(* IEC 61131-3 sources: ATCMcontrol_Engineering/src/COM/softing/fc/AddOns/Softing/4CPCTarget/Libs/ATCM_IEC1131_3/table_36, 9 files *)

(* ---- ctd.st ---- *)
(*[[
    UserURL= "ATCM:CTD_DINT.htm"
]]*)
(*
 *  IEC-1131-3 Standard Functionblock CTD for data type INT
 *  Purpose: Down Counter
 *)
FUNCTION_BLOCK CTD
VAR_INPUT  (* Inputs *)
    CD         : BOOL R_EDGE; (* count down if rising edge     *)
    LD         : BOOL;        (* if true, copy PV to CV        *)
    PV         : INT;         (* start value                   *)
END_VAR
VAR_OUTPUT (* Outputs *)
    Q          : BOOL;        (* TRUE if CV <= 0               *)
    CV         : INT;         (* counter output                *)
END_VAR

;(* add target specific implementation here *)

END_FUNCTION_BLOCK

(* ---- ctd_dint.st ---- *)
(*[[
    UserURL= "ATCM:CTD_DINT.htm"
]]*)
(*
 *  IEC-1131-3 Standard Functionblock CTD for data type DINT
 *  Purpose: Down Counter
 *)
FUNCTION_BLOCK CTD_DINT
VAR_INPUT  (* Inputs *)
    CD         : BOOL R_EDGE; (* count down if rising edge     *)
    LD         : BOOL;        (* if true, copy PV to CV        *)
    PV         : DINT;        (* start value                   *)
END_VAR
VAR_OUTPUT (* Outputs *)
    Q          : BOOL;        (* TRUE if CV <= 0               *)
    CV         : DINT;        (* counter output                *)
END_VAR

  IF LD THEN
	CV := PV;
  ELSIF CD AND (CV > FC_MIN_DINT) THEN
	CV:=CV-1;
  END_IF;

  Q := (CV <= 0);

END_FUNCTION_BLOCK

(* ---- ctd_dint_ex.st ---- *)
(*[[
    UserURL= "ATCM:CTD_DINT_EX.htm"
]]*)
(*
 *  IEC-1131-3 Standard Functionblock CTD for data type DINT
 *  Purpose: Down Counter with visualisation scaling parameters
 *)
FUNCTION_BLOCK CTD_DINT_EX
VAR_INPUT  (* Inputs *)
    CD         : BOOL R_EDGE; (* count down if rising edge     *)
    LD         : BOOL;        (* if true, copy PV to CV        *)
    PV         : DINT;        (* start value                   *)
END_VAR
VAR_INPUT  (* Parameters *)
    SCALEMIN   : DINT:=0;     (* minimum of scaling            *)
    SCALEMAX   : DINT:=100;   (* maximum of scaling            *)
END_VAR
VAR_OUTPUT (* Outputs *)
    Q          : BOOL;        (* TRUE if CV <= 0               *)
    CV         : DINT;        (* counter output                *)
    ERROR      : DINT;        (* error                         *)
END_VAR

ERROR := 0;
IF (SCALEMIN >= SCALEMAX) THEN
   ERROR:=-1;
END_IF;

IF LD THEN
   CV := PV;
ELSIF CD AND (CV > FC_MIN_DINT) THEN
   CV:=CV-1;
END_IF;

Q := (CV <= 0);

END_FUNCTION_BLOCK

(* ---- ctu.st ---- *)
(*[[
    UserURL= "ATCM:CTU_DINT.htm"
]]*)
(*
 *  IEC-1131-3 Standard Functionblock CTU for data type INT
 *  Purpose: Up Counter
 *)
FUNCTION_BLOCK CTU
VAR_INPUT (* Inputs *)
    CU         : BOOL R_EDGE; (* count up if rising edge *)
    R          : BOOL;        (* if true,  CV to zero    *)
    PV         : INT;         (* end value               *)
END_VAR
VAR_OUTPUT (* Outputs *)
    Q          : BOOL;        (* TRUE if CV >= PV        *)
    CV         : INT;         (* counter output          *)
END_VAR

;(* add target specific implementation here *)

END_FUNCTION_BLOCK

(* ---- ctu_dint.st ---- *)
(*[[
    UserURL= "ATCM:CTU_DINT.htm"
]]*)
(*
 *  IEC-1131-3 Standard Functionblock CTU for data type DINT
 *  Purpose: Up Counter
 *)
FUNCTION_BLOCK CTU_DINT
VAR_INPUT (* Inputs *)
    CU         : BOOL R_EDGE; (* count up if rising edge *)
    R          : BOOL;        (* if true,  CV to zero    *)
    PV         : DINT;        (* end value               *)
END_VAR
VAR_OUTPUT (* Outputs *)
    Q          : BOOL;        (* TRUE if CV >= PV        *)
    CV         : DINT;        (* counter output          *)
END_VAR

  IF R THEN
	CV := 0;
  ELSIF CU AND (CV < FC_MAX_DINT) THEN
	CV:=CV+1;
  END_IF;

  Q := (CV >= PV);

END_FUNCTION_BLOCK

(* ---- ctu_dint_ex.st ---- *)
(*[[
    UserURL= "ATCM:CTU_DINT_EX.htm"
]]*)
(*
 *  IEC-1131-3 Standard Functionblock CTU for data type DINT
 *  Purpose: Up Counter with visualisation scaling parameters
 *)
FUNCTION_BLOCK CTU_DINT_EX
VAR_INPUT  (* Inputs *)
    CU         : BOOL R_EDGE; (* count up if rising edge *)
    R          : BOOL;        (* if true,  CV to zero    *)
    PV         : DINT;        (* end value               *)
END_VAR
VAR_INPUT  (* Parameters *)
    SCALEMIN   : DINT:=0;     (* minimum of scaling      *)
    SCALEMAX   : DINT:=100;   (* maximum of scaling      *)
END_VAR
VAR_OUTPUT (* Outputs *)
    Q          : BOOL;        (* TRUE if CV >= PV        *)
    CV         : DINT;        (* counter output          *)
    ERROR      : DINT;        (* error                   *)
END_VAR

ERROR := 0;
IF (SCALEMIN >= SCALEMAX) THEN
    ERROR:=-1;
END_IF;

IF R THEN
    CV := 0;
ELSIF CU AND (CV < FC_MAX_DINT) THEN
    CV:=CV+1;
END_IF;

Q := (CV >= PV);

END_FUNCTION_BLOCK

(* ---- ctud.st ---- *)
(*[[
    UserURL= "ATCM:ctud_dint.htm"
]]*)
(*
 *  IEC-1131-3 Standard Functionblock CTUD for data type INT
 *  Purpose: Up/Down Counter
 *)
FUNCTION_BLOCK CTUD
VAR_INPUT (* Inputs *)
    CU         : BOOL R_EDGE; (* count up if rising edge   *)
    CD         : BOOL R_EDGE; (* count down if rising edge *)
    R          : BOOL;        (* Reset, set CV to 0        *)
    LD         : BOOL;        (* if true, copy PV to CV    *)
    PV         : INT;         (* start value               *)
END_VAR
VAR_OUTPUT (* Outputs *)
    QU         : BOOL;        (* TRUE if CV >= PV          *)
    QD         : BOOL;        (* TRUE if CV <= 0           *)
    CV         : INT;         (* counter output            *)
END_VAR

;(* add target specific implementation here *)

END_FUNCTION_BLOCK

(* ---- ctud_dint.st ---- *)
(*[[
    UserURL= "ATCM:CTUD_DINT.htm"
]]*)
(*
 *  IEC-1131-3 Standard Functionblock CTUD for data type DINT
 *  Purpose: Up/Down Counter
 *)
FUNCTION_BLOCK CTUD_DINT
VAR_INPUT (* Inputs *)
    CU         : BOOL R_EDGE; (* count up if rising edge   *)
    CD         : BOOL R_EDGE; (* count down if rising edge *)
    R          : BOOL;        (* Reset, set CV to 0        *)
    LD         : BOOL;        (* if true, copy PV to CV    *)
    PV         : DINT;        (* start value               *)
END_VAR
VAR_OUTPUT (* Outputs *)
    QU         : BOOL;        (* TRUE if CV >= PV          *)
    QD         : BOOL;        (* TRUE if CV <= 0           *)
    CV         : DINT;        (* counter output            *)
END_VAR

  IF R THEN
	CV := 0;
  ELSIF LD THEN
	CV := PV;
  ELSE
	IF NOT (CU AND CD) THEN
		IF CU AND (CV < FC_MAX_DINT) THEN
			CV:=CV+1;
		ELSIF CD AND (CV > FC_MIN_DINT) THEN
			CV := CV-1;
		END_IF;
	END_IF;
  END_IF;

  QU := (CV >= PV);
  QD := (CV <= 0);

END_FUNCTION_BLOCK

(* ---- ctud_dint_ex.st ---- *)
(*[[
    UserURL= "ATCM:CTUD_DINT_EX.htm"
]]*)
(*
 *  IEC-1131-3 Standard Functionblock CTUD for data type DINT
 *  Purpose: Up/Down Counter with visualisation scaling parameters
 *)
FUNCTION_BLOCK CTUD_DINT_EX
VAR_INPUT (* Inputs *)
    CU         : BOOL R_EDGE; (* count up if rising edge   *)
    CD         : BOOL R_EDGE; (* count down if rising edge *)
    R          : BOOL;        (* Reset, set CV to 0        *)
    LD         : BOOL;        (* if true, copy PV to CV    *)
    PV         : DINT;        (* start value               *)
END_VAR
VAR_INPUT (* Parameters *)
    SCALEMIN   : DINT:=0;     (* minimum of scaling *)
    SCALEMAX   : DINT:=100;   (* maximum of scaling *)
END_VAR
VAR_OUTPUT (* Outputs *)
    QU         : BOOL;        (* TRUE if CV >= PV   *)
    QD         : BOOL;        (* TRUE if CV <= 0    *)
    CV         : DINT;        (* counter output     *)
    ERROR      : DINT;        (* error              *)
END_VAR

ERROR := 0;
IF (SCALEMIN >= SCALEMAX) THEN
    ERROR:=-1;
END_IF;

IF R THEN
   CV := 0;
ELSIF LD THEN
   CV := PV;
ELSE
   IF NOT (CU AND CD) THEN
      IF CU AND (CV < FC_MAX_DINT) THEN
         CV:=CV+1;
      ELSIF CD AND (CV > FC_MIN_DINT) THEN
         CV := CV-1;
      END_IF;
   END_IF;
END_IF;

QU := (CV >= PV);
QD := (CV <= 0);

END_FUNCTION_BLOCK
